// TIA Portal project "Lab1_135" (V16)

(* hardware
DEVICE "S7-1200 station_1"  S7-1200 Station
   slot 0: "Rack_0"  S7-1200 Rack  Rack  V1.0
   slot 1: "PLC_1"  CPU 1214C DC/DC/DC  6ES7 214-1AG40-0XB0  V4.4
*)

// ===== PLC "PLC_1"  CPU 1214C DC/DC/DC =====

VAR_GLOBAL   // PLC tag table "Default tag table"
   "System_Byte" AT %MB800 : Byte;
   "FirstScan" AT %M800.0 : Bool;
   "DiagStatusUpdate" AT %M800.1 : Bool;
   "AlwaysTRUE" AT %M800.2 : Bool;
   "AlwaysFALSE" AT %M800.3 : Bool;
   "Clock_Byte" AT %MB801 : Byte;
   "Clock_10Hz" AT %M801.0 : Bool;
   "Clock_5Hz" AT %M801.1 : Bool;
   "Clock_2.5Hz" AT %M801.2 : Bool;
   "Clock_2Hz" AT %M801.3 : Bool;
   "Clock_1.25Hz" AT %M801.4 : Bool;
   "Clock_1Hz" AT %M801.5 : Bool;
   "Clock_0.625Hz" AT %M801.6 : Bool;
   "Clock_0.5Hz" AT %M801.7 : Bool;
   "Run" AT %I0.0 : Bool;
   "B_Run" AT %M0.0 : Bool;
   "Stop" AT %I0.1 : Bool;
   "Reset" AT %I0.2 : Bool;
   "B_Reset" AT %M0.1 : Bool;
   "Tag_2" AT %QB0 : Byte;
   "Pulse1" AT %M3.0 : Bool;
   "B_SHR_L" AT %M0.2 : Bool;
   "Pulse2" AT %M3.1 : Bool;
   "Tag_3" AT %Q0.0 : Bool;
   "Tag_4(1)" AT %Q0.1 : Bool;
   "Tag_5" AT %Q0.2 : Bool;
   "Tag_6" AT %Q0.3 : Bool;
   "Tag_7" AT %Q0.4 : Bool;
   "Tag_8" AT %Q0.5 : Bool;
   "Tag_9" AT %Q0.6 : Bool;
   "Tag_4" AT %Q0.7 : Bool;
END_VAR

// folder: System blocks/Program resources

DATA_BLOCK "Timer1"   // DB1
{ S7_Optimized_Access := 'TRUE' }
AUTHOR : Simatic
FAMILY : IEC
NAME : IEC_TMR
VERSION : 1.0
// stored: InstanceOfName IEC_TIMER
"IEC_TIMER"
BEGIN
END_DATA_BLOCK

DATA_BLOCK "Timer2"   // DB2
{ S7_Optimized_Access := 'TRUE' }
AUTHOR : Simatic
FAMILY : IEC
NAME : IEC_TMR
VERSION : 1.0
// stored: InstanceOfName IEC_TIMER
"IEC_TIMER"
BEGIN
END_DATA_BLOCK

// folder: (top level)

ORGANIZATION_BLOCK "Main"   // OB1, LAD, ProgramCycle
TITLE = "Main Program Sweep (Cycle)"
{ S7_Optimized_Access := 'TRUE' }
VERSION : 0.1
   VAR_INPUT
      Initial_Call : Bool;   // Initial call of this OB
      Remanence : Bool;   // =True, if remanent data are available
   END_VAR
   VAR_TEMP   // added for the SCL form of the ladder/FBD networks
      _w1 : Bool;
   END_VAR
BEGIN

REGION Network 1
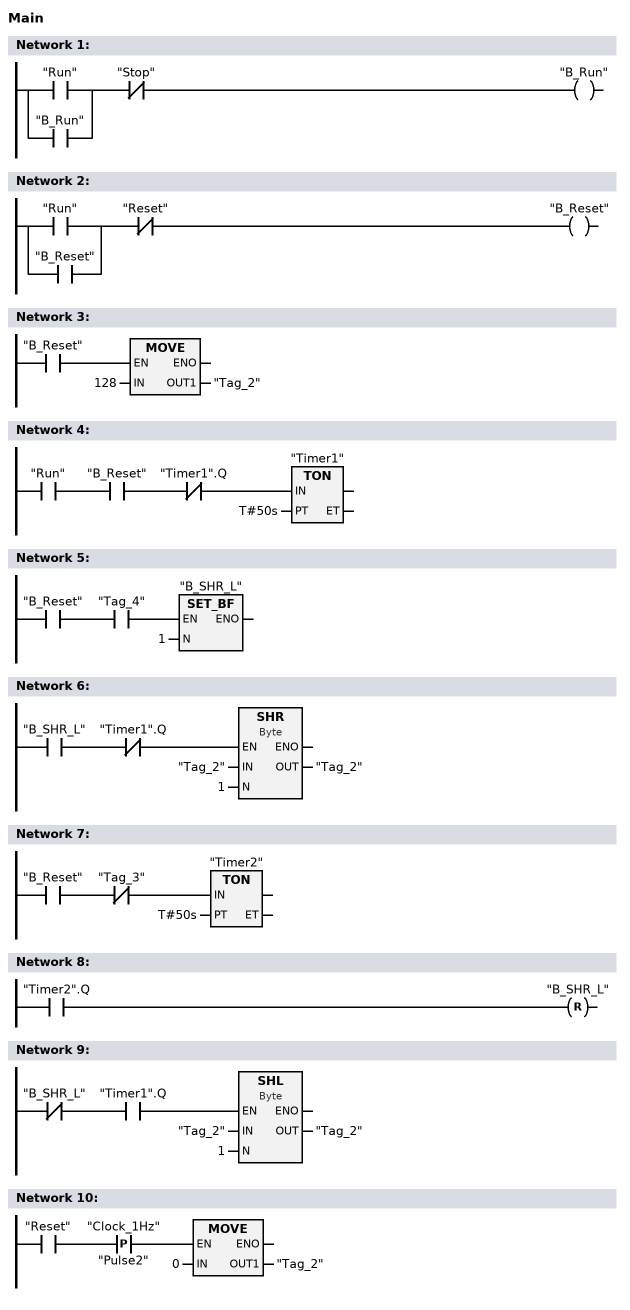
   RUNG wire#powerrail
      Contact( "Run" )
      wire#w1
      I_Contact( "Stop" )
      Coil( "B_Run" )
   END_RUNG
   RUNG wire#powerrail
      Contact( "B_Run" )
   END_RUNG wire#w1
   // the same network as SCL:
   "B_Run" := ("Run" OR "B_Run") AND NOT "Stop";
END_REGION

REGION Network 2
   RUNG wire#powerrail
      Contact( "Run" )
      wire#w1
      I_Contact( "Reset" )
      Coil( "B_Reset" )
   END_RUNG
   RUNG wire#powerrail
      Contact( "B_Reset" )
   END_RUNG wire#w1
   // the same network as SCL:
   "B_Reset" := ("Run" OR "B_Reset") AND NOT "Reset";
END_REGION

REGION Network 3
   RUNG wire#powerrail
      Contact( "B_Reset" )
      Move(in := 128, out1 => "Tag_2")
   END_RUNG
   // the same network as SCL:
   IF "B_Reset" THEN "Tag_2" := 128; END_IF;
END_REGION

REGION Network 4
   "Timer1".TON(IN := "Run" AND "B_Reset" AND NOT "Timer1".Q, PT := T#50s);
END_REGION

REGION Network 5
   // no SCL statement known for SBitfield: written as a call
   IF "B_Reset" AND "Tag_4" THEN SET_BF(operand := "B_SHR_L", n := 1); END_IF;
END_REGION

REGION Network 6
   RUNG wire#powerrail
      Contact( "B_SHR_L" )
      I_Contact( "Timer1".Q )
      { S7_Templates := "SrcType := Byte" } Shr(in := "Tag_2", n := 1, out => "Tag_2")
   END_RUNG
   // the same network as SCL:
   IF "B_SHR_L" AND NOT "Timer1".Q THEN "Tag_2" := SHR(IN := "Tag_2", N := 1); END_IF;
END_REGION

REGION Network 7
   "Timer2".TON(IN := "B_Reset" AND NOT "Tag_3", PT := T#50s);
END_REGION

REGION Network 8
   RUNG wire#powerrail
      Contact( "Timer2".Q )
      R_Coil( "B_SHR_L" )
   END_RUNG
   // the same network as SCL:
   IF "Timer2".Q THEN "B_SHR_L" := FALSE; END_IF;
END_REGION

REGION Network 9
   RUNG wire#powerrail
      I_Contact( "B_SHR_L" )
      Contact( "Timer1".Q )
      { S7_Templates := "SrcType := Byte" } Shl(in := "Tag_2", n := 1, out => "Tag_2")
   END_RUNG
   // the same network as SCL:
   IF NOT "B_SHR_L" AND "Timer1".Q THEN "Tag_2" := SHL(IN := "Tag_2", N := 1); END_IF;
END_REGION

REGION Network 10
   RUNG wire#powerrail
      Contact( "Reset" )
      P_Contact(operand := "Clock_1Hz", bit := "Pulse2")
      Move(in := 0, out1 => "Tag_2")
   END_RUNG
   // the same network as SCL:
   #_w1 := "Reset" AND "Clock_1Hz" AND NOT "Pulse2";   // rising edge of "Clock_1Hz"
   "Pulse2" := "Clock_1Hz";
   IF #_w1 THEN "Tag_2" := 0; END_IF;
END_REGION
END_ORGANIZATION_BLOCK